{attribute 'qualified_only'}
{attribute 'strict'}
{attribute 'to_string'}
TYPE TExecutionState :
(	
	Unknown := 0,
	Ready,
    Starting,
    Busy,
	Error,
	Warning
);
END_TYPE

(* stored: Version 1.1.0.1, ProductVersion 3.1.4024.12
   DUT TExecutionState: Id {0bd3fd33-8d05-43c8-9593-8d1d7adee12a} *)
